Universal Robots PolyScope program: d_full_up.urp

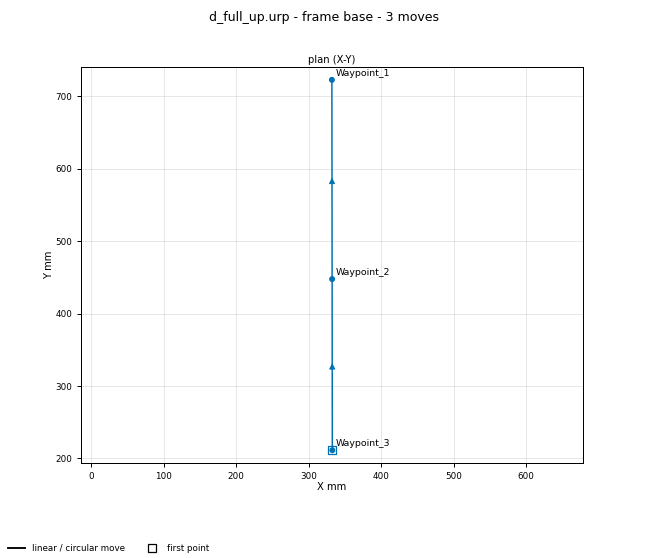
[picture p0: tool path of d_full_up.urp in frame base, 3 of 3 moves have a stored position in this frame; points joined in program order, loops and branches not executed]
Program d_full_up (installation=string_planes directory=/programs createdIn=5.17.3 lastSavedIn=5.17.3 robotSerialNumber=20245501435)
Calibrated DH parameters: a=[0.000154, -0.137004, -0.385524, -0.00002, 0.000092, 0]; d=[0.162441, 211.794786, -230.585024, 18.923638, 0.099786, 0.09951]; alpha=[1.569493, -0.001902, 0.003874, 1.570111, -1.570167, 0]; deltaTheta=[0, -1.242934, 1.056292, 0.186646, 0.000002, 0.000001]
InitVariablesNode
Robot Program (runOnlyOnce=false)
  MoveL speed 250 mm/s, acceleration 1200 mm/s^2 (useActiveTCP=true) feature=Joint_6_name
    Waypoint Waypoint_3: TCP in base x=332.581 y=211.38 z=108.291 mm, rx=-1.645 ry=-2.1081 rz=1.0591 rad; joints [-171.842, -51.824, 127.067, -122.03, -106.624, -178.984] deg; TCP offset x=28.21 y=-96.107 z=-99.69 mm, rx=0 ry=0 rz=0 rad; feature pose in base x=332.588 y=211.391 z=108.297 mm, rx=-1.6449 ry=-2.1082 rz=1.0591 rad
    Waypoint Waypoint_2: motionParameters(blendRadius=0.05); TCP in base x=332.299 y=447.473 z=108.291 mm, rx=-1.645 ry=-2.1081 rz=1.0591 rad; joints [-146.713, -43.689, 102.49, -103.08, -88.878, -161.003] deg; feature pose in base x=332.293 y=447.486 z=108.291 mm, rx=-1.645 ry=-2.1081 rz=1.0591 rad
    Waypoint Waypoint_1: TCP in base x=331.971 y=722.315 z=108.291 mm, rx=-1.645 ry=-2.1081 rz=1.0591 rad; joints [-129.709, -21.469, 51.981, -76.268, -76.862, -148.975] deg; feature pose in base x=331.955 y=722.33 z=108.302 mm, rx=-1.645 ry=-2.1081 rz=1.0591 rad
